TYPE _ST_Timestamp :
STRUCT
	nSeconds : LINT;
	nNanoseconds : DINT;
END_STRUCT
END_TYPE

(* stored: Version 1.1.0.1
   DUT _ST_Timestamp: Id {01de8f73-6f27-4d69-8664-6f5026c4f720} *)
